// TIA Portal V19 export
VAR_GLOBAL   // PLC tag table "Default tag table"
   "System_Byte(1)" AT %MB1 : Byte;
   "Clock_Byte(1)" AT %MB0 : Byte;
   "Clock_10Hz(1)" AT %M0.0 : Bool;
   "Clock_5Hz(1)" AT %M0.1 : Bool;
   "Clock_2.5Hz(1)" AT %M0.2 : Bool;
   "Clock_2Hz(1)" AT %M0.3 : Bool;
   "Clock_1.25Hz(1)" AT %M0.4 : Bool;
   "Clock_1Hz(1)" AT %M0.5 : Bool;
   "Clock_0.625Hz(1)" AT %M0.6 : Bool;
   "Clock_0.5Hz(1)" AT %M0.7 : Bool;
END_VAR
